INTERFACE ITF_CylinderBase//cylinder no feedback spring return solonoid

METHOD Extend : BOOL
END_METHOD

PROPERTY Extended : BOOL	//Status bit for the position of the cylinder
GET
END_GET
END_PROPERTY

PROPERTY Extending : BOOL
GET
END_GET
END_PROPERTY

PROPERTY ExtendTime : TIME	//Approximate expected time for the cylinder to complete an extension cycle
GET
END_GET
SET
END_SET
END_PROPERTY

METHOD Idle : BOOL
END_METHOD

METHOD Retract : UDINT
END_METHOD

PROPERTY Retracted : BOOL	//Status bit for the position of the cylinder
GET
END_GET
END_PROPERTY

PROPERTY Retracting : BOOL
GET
END_GET
END_PROPERTY

PROPERTY RetractTime : TIME
GET
END_GET
SET
END_SET
END_PROPERTY

PROPERTY TimeoutFactor : LREAL	//Multiplicative factor that determines error timeout threshold based on the expected time
GET
END_GET
SET
END_SET
END_PROPERTY

END_INTERFACE

(* stored: Version 1.1.0.1, ProductVersion 3.1.4024.10
   Itf ITF_CylinderBase: Id {341131b4-468e-42eb-a6b0-a67dca0a8688}
   Folder 01_Properties: Id {b6a350b3-87a9-4d94-952f-1d746bcd503d}
   Folder 01_Config: Id {43a174e4-ccf3-49be-8e8c-146032af8800}
   Folder 02_Control: Id {1e5282f1-6dff-45c7-bb6f-96cac7da5a39}
   Folder 03_Status: Id {afd777e9-1f1e-43fa-9ccc-b9eb9d2a3a1b}
   Folder 02_Methods: Id {7ef57548-ebf5-4dae-a304-a8844e6fa8af}
   Method Extend: Id {23114865-3a0a-4898-bc94-e9562cf85b65}
   Property Extended: Id {f239fb64-1f4c-4854-b9dc-dea4835573b5}
   Get Get: Id {3e340c65-b28a-4a76-9824-ce0f037495b2}
   Property Extending: Id {991b3c75-876a-4f07-a927-a3a3ea0b3ede}
   Get Get: Id {e49d3421-234f-4d1d-adf6-676173172884}
   Property ExtendTime: Id {229c5001-0fdb-45dc-b199-d24b538b4c46}
   Get Get: Id {f4c53921-cd1c-4b42-a088-c948868e9275}
   Set Set: Id {233fb3b0-f71f-440d-b15c-e6c53fe1281b}
   Method Idle: Id {c7472d65-1ed8-4ddb-8643-1f39e3a47e0c}
   Method Retract: Id {85beeaa7-d2e5-41e1-a561-42650b31a0ca}
   Property Retracted: Id {00c8c591-312a-47ea-b899-eed50767d7ca}
   Get Get: Id {831fa028-4389-4686-9765-557c4b2778ea}
   Property Retracting: Id {8d6531d6-baa8-4b01-8fa5-3a596d55e4bd}
   Get Get: Id {49669248-45e1-45d1-a256-fe80773e8ee5}
   Property RetractTime: Id {2c44d9cd-557a-4cff-8038-4f37db9f471f}
   Get Get: Id {21517817-ef43-4cf8-a3ac-ca2746ba5990}
   Set Set: Id {791cf7ca-1565-4a2c-a8c9-cb7c43406c01}
   Property TimeoutFactor: Id {8658084e-739d-4edf-b642-c29237f14bec}
   Get Get: Id {7eebbbde-d8e9-4b76-8570-88dcd2d7c23a}
   Set Set: Id {395b3a8d-458c-450c-afe3-681325d327e6} *)
